// SIMATIC S7-200 project (STEP 7-Micro/WIN), CPU 222 REL 02.01

SYMBOL_TABLE USER1
E0               M0.0     // Etapa 0
E1               M0.1     // Etapa 1
E2               M0.2     // Etapa 2
E3               M0.3     // Etapa 3
E4               M0.4     // Etapa 4
E5               M0.5     // Etapa 5
E6               M0.6     // Etapa 6
E7               M0.7     // Etapa 7
E8               M1.0     // Etapa 8
SR1              I0.1     // Sensor de posição de recuo atuador 1
SR2              I0.2     // Sensor de posição de recuo atuador 2
BI               I0.6     // Botão de inicio
SA1              I0.3     // Sensor de posição do avanço 1
Temp_1           T37      // Temporizador de 3s
SA2              I0.4     // Sensor posição de avanço 2
Temp_2           T38      // Temporizador de 10s
BT               I0.7     // Botão inicio 2
RECOLHE          I0.5     // Botão recolhe
Y1               Q0.1     // Avanço atuador 1
Y2               Q0.0     // Recuo do atuador 1
Y3               Q0.3     // Avanço atuador 2
Y4               Q0.2     // Recuo do atuador 2
SL               Q0.4     // Sinal luminoso de interrupção
END_SYMBOL_TABLE

ORGANIZATION_BLOCK MAIN:OB1
TITLE=PROGRAM COMMENTS
BEGIN
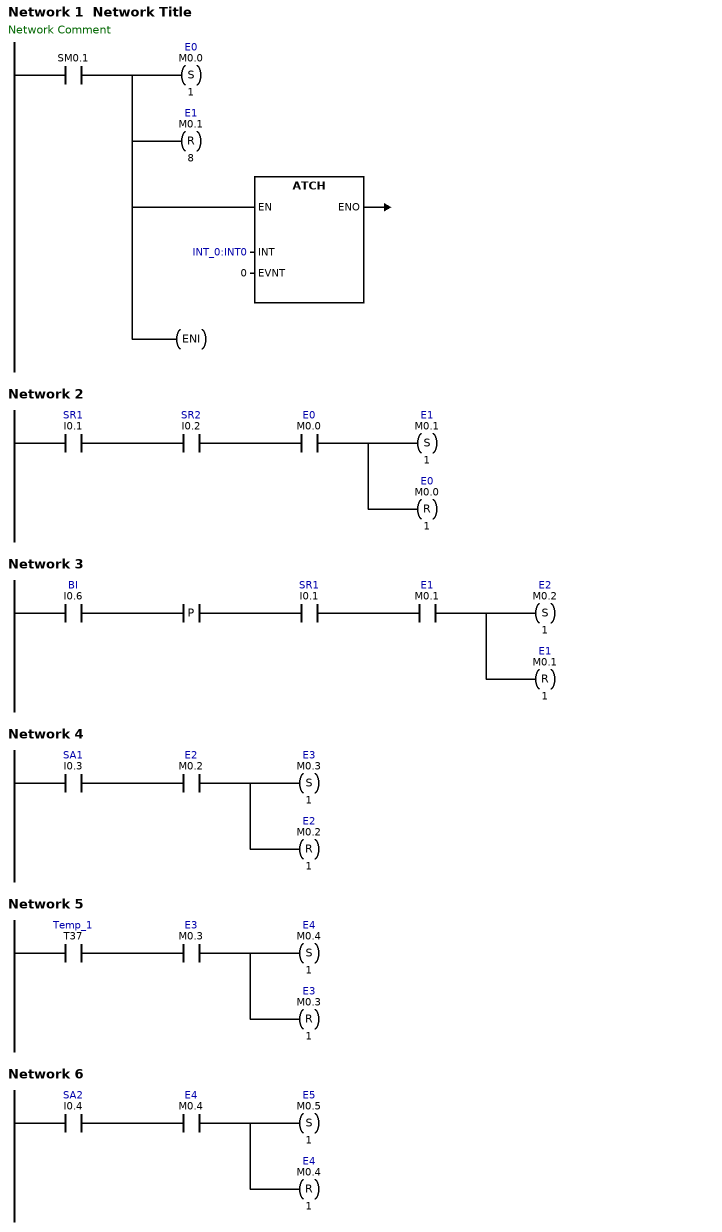
Network 1 // Network Title
// Network Comment
LD     SM0.1
S      E0:M0.0, 1
R      E1:M0.1, 8
ATCH   INT_0:INT0, 0
ENI
Network 2
LD     SR1:I0.1
A      SR2:I0.2
A      E0:M0.0
S      E1:M0.1, 1
R      E0:M0.0, 1
Network 3
LD     BI:I0.6
EU
A      SR1:I0.1
A      E1:M0.1
S      E2:M0.2, 1
R      E1:M0.1, 1
Network 4
LD     SA1:I0.3
A      E2:M0.2
S      E3:M0.3, 1
R      E2:M0.2, 1
Network 5
LD     Temp_1:T37
A      E3:M0.3
S      E4:M0.4, 1
R      E3:M0.3, 1
Network 6
LD     SA2:I0.4
A      E4:M0.4
S      E5:M0.5, 1
R      E4:M0.4, 1
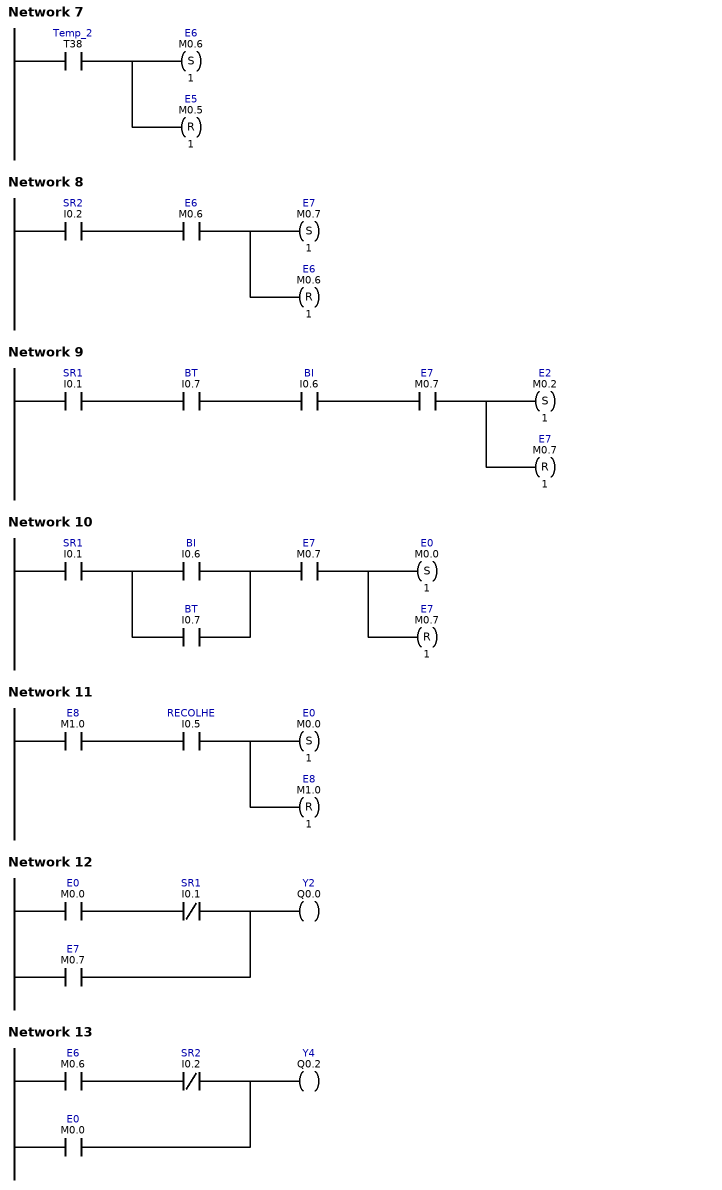
Network 7
LD     Temp_2:T38
S      E6:M0.6, 1
R      E5:M0.5, 1
Network 8
LD     SR2:I0.2
A      E6:M0.6
S      E7:M0.7, 1
R      E6:M0.6, 1
Network 9
LD     SR1:I0.1
A      BT:I0.7
A      BI:I0.6
A      E7:M0.7
S      E2:M0.2, 1
R      E7:M0.7, 1
Network 10
LD     SR1:I0.1
LD     BI:I0.6
O      BT:I0.7
ALD
A      E7:M0.7
S      E0:M0.0, 1
R      E7:M0.7, 1
Network 11
LD     E8:M1.0
A      RECOLHE:I0.5
S      E0:M0.0, 1
R      E8:M1.0, 1
Network 12
// (network saved uncompiled; LAD cells follow)
// row 0: c0 -| |- E0:M0.0  c1 -|/|- SR1:I0.1 v  c2 -( ) Y2:Q0.0
// row 1: c0 -| |- E7:M0.7  c1 -- ^
Network 13
// (network saved uncompiled; LAD cells follow)
// row 0: c0 -| |- E6:M0.6  c1 -|/|- SR2:I0.2 v  c2 -( ) Y4:Q0.2
// row 1: c0 -| |- E0:M0.0  c1 -- ^
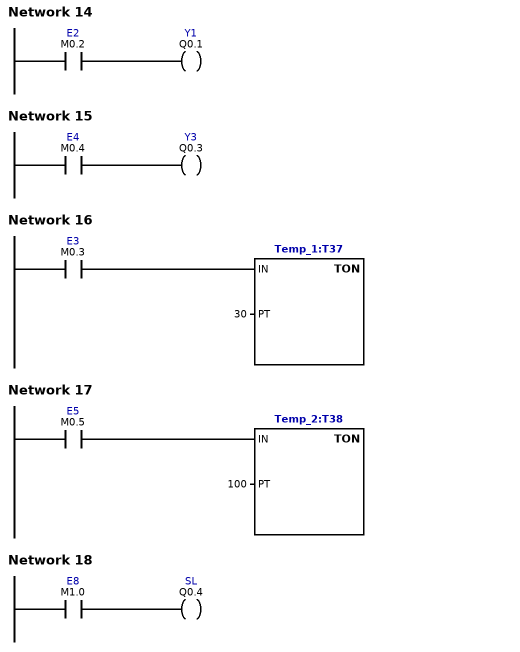
Network 14
// (network saved uncompiled; LAD cells follow)
// row 0: c0 -| |- E2:M0.2  c1 -( ) Y1:Q0.1
Network 15
// (network saved uncompiled; LAD cells follow)
// row 0: c0 -| |- E4:M0.4  c1 -( ) Y3:Q0.3
Network 16
LD     E3:M0.3
TON    Temp_1:T37, 30
Network 17
LD     E5:M0.5
TON    Temp_2:T38, 100
Network 18
LD     E8:M1.0
=      SL:Q0.4
END_ORGANIZATION_BLOCK

INTERRUPT_BLOCK INT_0:INT0
TITLE=INTERRUPT ROUTINE COMMENTS
BEGIN
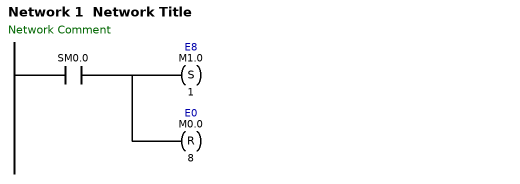
Network 1 // Network Title
// Network Comment
LD     SM0.0
S      E8:M1.0, 1
R      E0:M0.0, 8
END_INTERRUPT_BLOCK
